KUKA KRL data list: CVExample.dat

&ACCESS RVO
&REL 1
&PARAM EDITMASK = *
&PARAM TEMPLATE = C:\KRC\Roboter\Template\ExpertVorgabe
DEFDAT CVExample PUBLIC

int myvar = 123456879

ENDDAT
